TYPE ST_MasterCTRL :
STRUCT
	

	// Request Flags
	bManualModeRequest					:BOOL;
	
	bCycleStopRequest					:BOOL;
	
	bNoImmediateFault					:BOOL;
	bNoCycleStopFault					:BOOL;


	// Feedback Flags
	bAllStationsReady					:BOOL;
	bAllStationsStopped					:BOOL;
	
	bPowerUpTimerComplete				:BOOL;

	
//-------------------------------------------------------------------------------oldschoo1
		
END_STRUCT
END_TYPE

(* stored: Version 1.1.0.1, ProductVersion 3.1.4024.13
   DUT ST_MasterCTRL: Id {0cf524b1-b3b8-486a-882b-6a9427e24a47} *)
